// PORTED. Pins the wall-clock deadline, which had no coverage at all in the
// original verifier (R14) - only the cycle budget was exercised.
//
// The inner test never finishes, so only a deadline can end it. Its CYCLE budget
// is set to zero so the wall clock is unambiguously what fired; without that, at a
// fast task period a cycle budget could expire first and the test would pass for
// the wrong reason.
//
// The second assertion is the one that matters: the failure must NAME the wall
// clock. A deadline that fires correctly but says the wrong thing is still a
// defect - the message is what someone reads at three in the morning.
FUNCTION_BLOCK CHAR_WallClockTimeout IMPLEMENTS I_Test
VAR
	Inner	 : TestSuite<4>;
	Recorder : RecordingReporter;
	Budgets	 : ST_TestBudgets;
	Phase	 : DINT;
	Scans	 : DINT;
	Spinner : HangingBodyTest;
	ExpectedCount : UDINT;
	ActualCount	  : UDINT;
END_VAR

METHOD Run : BOOL
VAR_INPUT
	Enable : BOOL;
	Test   : I_TestAssertions;
END_VAR
Scans := Scans + 1;
IF Scans > 500 THEN
	Test.Fail('the inner suite never completed');
	Run := TRUE;
	RETURN;
END_IF

CASE Phase OF

0:
	// Zero disables the scan budget. Explicitly SET, not merely left alone - an
	// unset field inherits the suite default instead of disabling anything.
	Budgets.Body.Cycles		  := 0;
	Budgets.Body.IsCyclesSet  := TRUE;
	Budgets.Body.Timeout	  := T#200MS;
	Budgets.Body.IsTimeoutSet := TRUE;

	Inner.SetLabel('CHAR_WallClock_Subject');
	Inner.AddReporter(Recorder);
	Inner.Register(Spinner, 'Spinner', Budgets);
	Phase := 1;
	Run	  := FALSE;

1:
	IF Inner.Run(Enable := TRUE) THEN
		Phase := 2;
	END_IF
	Run := FALSE;

2:
	ExpectedCount := 1;
	ActualCount	  := Recorder.StatFailures;
	Test.AssertEqual(ExpectedCount, ActualCount, 'the spinning test failed');

	Test.AssertTrue(Recorder.CaseFailureKind('Spinner') = E_FailureKind.Timeout,
					'and failed as a timeout');

	Test.AssertTrue(Recorder.FailureContains('Spinner', 'wall time'),
					'the failure names the wall-clock deadline');

	Run := TRUE;

END_CASE
END_METHOD

END_FUNCTION_BLOCK

(* stored: Version 1.1.0.1, ProductVersion 3.1.4026.18
   POU CHAR_WallClockTimeout: Id {57fbfd8a-8cfe-412b-8c7c-2a96f33fbfe5}, SpecialFunc None
   Folder I_Test: Id {cca1a501-80ad-4fdb-976a-7d06af68525a}
   Method Run: Id {e3a70411-75e2-4cc6-b80f-1fde40a1dd62} *)
